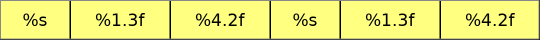
VISUALIZATION VISU_CONFIG_LIGNE_GAZ_SEUIL_MFC_MKS  // 540x40
VAR_IN_OUT
	m_Input_MASSFLOW:		BLOCK_MFC_MKS_NoCoE;
END_VAR
    Rectangle (70,0 100x40), "%1.3f", text variable: m_Input_MASSFLOW.CONF_Nom_Coef, input disabled if: NOT Global_Variables.PRG_USER.ACTU_USER.CONF_MACHINE
        OnMouseDown: write the text variable via Edit
    Rectangle (170,0 100x40), "%4.2f", text variable: m_Input_MASSFLOW.CONF_Nom_max_flow, input disabled if: NOT Global_Variables.PRG_USER.ACTU_USER.CONF_MACHINE
        OnMouseDown: write the text variable via VisuDialogs.Numpad
    Rectangle (340,0 100x40), "%1.3f", text variable: m_Input_MASSFLOW.CONF_Util_Coef, input disabled if: NOT Global_Variables.PRG_USER.ACTU_USER.CONF_MACHINE
        OnMouseDown: write the text variable via VisuDialogs.Numpad
    Rectangle (440,0 100x40), "%4.2f", text variable: m_Input_MASSFLOW.CONF_Util_Max_Flow, input disabled if: NOT Global_Variables.PRG_USER.ACTU_USER.CONF_MACHINE
    Rectangle (0,0 70x40), "%s", text variable: m_Input_MASSFLOW.CONF_Nom_Name, input disabled if: NOT Global_Variables.PRG_USER.ACTU_USER.CONF_MACHINE
        OnMouseDown: write the text variable via VisuDialogs.Keypad
    Rectangle (270,0 70x40), "%s", text variable: m_Input_MASSFLOW.CONF_Util_Name, input disabled if: NOT Global_Variables.PRG_USER.ACTU_USER.CONF_MACHINE
        OnMouseDown: write the text variable via VisuDialogs.Keypad
END_VISUALIZATION

(* stored: Version 1.1.0.1, ProductVersion 3.1.4024.6
   Visu VISU_CONFIG_LIGNE_GAZ_SEUIL_MFC_MKS: Id {2801655a-4d7f-430c-8782-120c51f62d4e} *)
